FUNCTION GetCycleTimeInSeconds : LREAL
VAR CONSTANT
	DefaultCTUnit : LREAL := 0.0000001; // PlcTaskSystemInfo.CycleTime is in [100*ns]
END_VAR
VAR
	cycleTime : UDINT;
END_VAR

cycleTime := _TaskInfo[GETCURTASKINDEXEX()].CycleTime;
GetCycleTimeInSeconds := TO_LREAL(cycleTime) * DefaultCTUnit;

END_FUNCTION

(* stored: Version 1.1.0.1
   POU GetCycleTimeInSeconds: Id {dfc608dd-d47c-054c-06a3-41bbea9aa324}, SpecialFunc None *)
